(* PLC project Tc2_Standard.WLEN Demo, tc3-libraries-kb TwinCAT 3.1 *)
(* stored: creationDateTime 2026-05-10T08:00:00, modificationDateTime 2026-05-10T08:00:00 *)

PROGRAM P_Demo_WLEN
  VAR
    sResult : INT;  (* WLEN 的返回值（监视） *)
    bRun : BOOL;  (* 触发一次 WLEN 调用 *)
  END_VAR

            // ============================================================
// Tc2_Standard.WLEN 演示程序（FUNCTION）
// ============================================================
// 场景：对 WSTRING 执行 LEN 操作
// 验证步骤：
//   1. 编译并登录目标
//   2. 强制 bRun := TRUE 一个周期
//   3. 观察 sResult = 4
//   4. bRun 自动复位
// ============================================================

IF bRun THEN
    sResult := WLEN("SUSI");
    bRun := FALSE;
END_IF;

          
END_PROGRAM
